{attribute 'hide_all_locals'}
FUNCTION_BLOCK RemoveAllMoverFromGroup IMPLEMENTS ITask
VAR_INPUT
END_VAR
VAR_OUTPUT
END_VAR
VAR
	RemoveAllFromGrp			: MC_UngroupAllAxes;
	_caGroup			: ICollisionGroup;
	State: INT;
	_removeAllMovers : BOOL;
	_busy : BOOL;
	_error : BOOL;
	_done : BOOL;
	_moverNumber : INT;
END_VAR

CASE State OF
	0:
		IF _removeAllMovers THEN
			_done := FALSE;
			_error := FALSE;
			_busy := TRUE;
			RemoveAllFromGrp.Execute := TRUE;
			IF RemoveAllFromGrp.Busy THEN
				_removeAllMovers := FALSE;
				State := 10;
			END_IF
		END_IF
		
	10:
		IF NOT RemoveAllFromGrp.Busy THEN
			IF RemoveAllFromGrp.Done THEN
				_done := TRUE;
			ELSIF RemoveAllFromGrp.Error THEN
				_error := TRUE;
			END_IF
			_busy := FALSE;
			RemoveAllFromGrp.Execute := false;
			State := 0;
		END_IF
END_CASE


RemoveAllFromGrp(AxesGroup := _caGroup.GroupRef);

METHOD Abort : BOOL
RemoveAllFromGrp.Execute := FALSE;
Abort := true;
State := 0;
END_METHOD


PROPERTY Busy : BOOL
GET
Busy := _busy;
END_GET
END_PROPERTY


PROPERTY Done : BOOL
GET
Done := _done;
END_GET
END_PROPERTY


PROPERTY Error : BOOL
GET
Error := _error;
END_GET
END_PROPERTY

METHOD FB_init : BOOL
VAR_INPUT
	bInitRetains : BOOL; // if TRUE, the retain variables are initialized (warm start / cold start)
	bInCopyCode : BOOL;  // if TRUE, the instance afterwards gets moved into the copy code (online change)
	CAGroup : ICollisionGroup;	
END_VAR
_caGroup := CAGroup;
END_METHOD

METHOD RemoveAllMover : BOOL
RemoveAllMover := _removeAllMovers := true;
END_METHOD

END_FUNCTION_BLOCK

(* stored: Version 1.1.0.1, ProductVersion 3.1.4024.9
   POU RemoveAllMoverFromGroup: Id {894ab397-c87f-4d26-bea3-6776a2e45544}, SpecialFunc None
   Method Abort: Id {a22f45bd-5352-4828-a3a0-02009b309eee}
   Property Busy: Id {aa2b0c68-97ac-4e3d-8af8-744ea2020f28}
   Get Get: Id {4e86423a-4aac-40b3-b4a2-8c9b974f971d}
   Property Done: Id {61a22672-181b-4578-b9cc-2097dc895769}
   Get Get: Id {4047a176-4d61-4706-a4a7-25e0a91951a2}
   Property Error: Id {cf277637-4844-4a07-9169-02da751dae99}
   Get Get: Id {58e25449-64dd-43cb-bed2-688efb8d28f8}
   Method FB_init: Id {4e9b5adb-fcc3-45b9-baf7-0b8c71d28b86}
   Method RemoveAllMover: Id {9cf1b53b-0b00-45d8-9017-648dead49a6a} *)
